{attribute 'qualified_only'}
VAR_GLOBAL CONSTANT

    NUM_MOVERS   : USINT := 4;    // This should be set to the exact number of movers on the system
    NUM_STATIONS : USINT := 5;    // This should be set to a value equal to or greater than the number of stations needed
    TRACK_LENGTH : LREAL := 1500; // This should be set to the exact length [mm] of the track system
	
    {attribute 'TcInitSymbol'}
    pXtsProcessingUnit : OTCID:=0; // This pointer needs to be initialized in the Main Instance, under Symbol Initialization

	NUM_TRACKS  : USINT := 1;	// This is the number of logical tracks in the system

	
		
END_VAR
VAR_GLOBAL
	newCallTime: LREAL;
	order_number : INT :=1;
	
END_VAR

(* stored: Version 1.1.0.1, ProductVersion 3.1.4024.13
   GVL GVL: Id {ba655886-9947-4787-bd10-a16d0603440f} *)
